// TIA Portal V20 export
DATA_BLOCK "PM07"   // DB333
// stored: MemoryReserve 100
   VAR
      "JR WINDER CLAMP TOP REAR  UP" : Bool := FALSE;
      "JR WINDER CLAMP TOP REAR  DOWN" : Bool := FALSE;
      "JR WINDER CLAMP BTM REAR UP" : Bool := FALSE;
      "JR WINDER CLAMP BTM REAR DOWN" : Bool := FALSE;
      "JR WINDER CLAMP TOP FRONT UP" : Bool := FALSE;
      "JR WINDER CLAMP TOP FRONT DOWN" : Bool := FALSE;
      "JR WINDER CLAMP BTM FRONT UP" : Bool := FALSE;
      "JR WINDER CLAMP BTM FRONT DOWN" : Bool := FALSE;
      SPARE : Bool := FALSE;
      SPARE_1 : Bool := FALSE;
      "PUSH ROLLER FORWARD" : Bool := FALSE;
      "PUSH ROLLER BACKWARD" : Bool := FALSE;
      "ANODE CONVEYOR COVER FORWARD" : Bool := FALSE;
      "ANODE CONVEYOR COVER BACKWARD" : Bool := FALSE;
      "CATHODE CONVEYOR COVER FORWARD" : Bool := FALSE;
      "CATHODE CONVEYOR COVER BACKWARD" : Bool := FALSE;
   END_VAR
BEGIN
END_DATA_BLOCK
